# EPICS autosave request: tests/testfiles/cfg/SF_OpticsMSEX_PV.req
$(SYS):ONOFF
$(SYS):K2L-SET
